{region '#Template'}
	{attribute 'Version' := '5.0.0.0'}
	{attribute 'Tags' := '"LCID": "1031", "Text": "AC, Allgemein, AHU, Betriebsart"'}
	{attribute 'Tags' := '"LCID": "1033", "Text": "AC, General, AHU, Operating mode"'}
	{attribute 'Using' := '"Type": "Template", "URI": "E_BA_AC_OpMod01"'}
	{attribute 'Using' := '"Type": "Template", "URI": "E_BA_OnOffA"'}
	{attribute 'Using' := '"Type": "Template", "URI": "E_BA_OnOff"'}
	{attribute 'Description' := '"LCID": "1031", "Text": "Betriebsart"'}
	{attribute 'Description' := '"LCID": "1033", "Text": "Operating mode"'}
{endregion}
FUNCTION_BLOCK FB_BA_AC_OpMod1St EXTENDS FB_BA_View
VAR_INPUT
	bSmExttSuA				: BOOL;	// smoke extraction supply air
	bSmExttExhA				: BOOL;	// smoke extraction exhaust air
	bFireDetc				: BOOL;	// fire detection alarm
	bForcVent				: BOOL;	// Forced ventilation
	bEmgOff					: BOOL;	// emergency stop
	bFrst					: BOOL;	// Frost protection is active
	bCentSwiOff				: BOOL;	// Central switch-off	
	bAlmShutOff				: BOOL;	// Shut Off plant collective alarm
	bNgtCol					: BOOL;	// Summer night cooling
	bColDwnPrtc				: BOOL;	// Cooling down protection
	bOvrHtgPrtc				: BOOL;	// Overheating protection
END_VAR
VAR_OUTPUT
	eOpMode					: E_BA_AC_OpMod01;
END_VAR
VAR_INPUT CONSTANT
	OpModMan				: FB_BA_MV_Op;	
	Sched					: FB_BA_SchedM;
	OpModPr					: FB_BA_MV_Op;
END_VAR
VAR
	PrioSwiOpMod			: FB_BA_PrioSwi_UDI24;
END_VAR

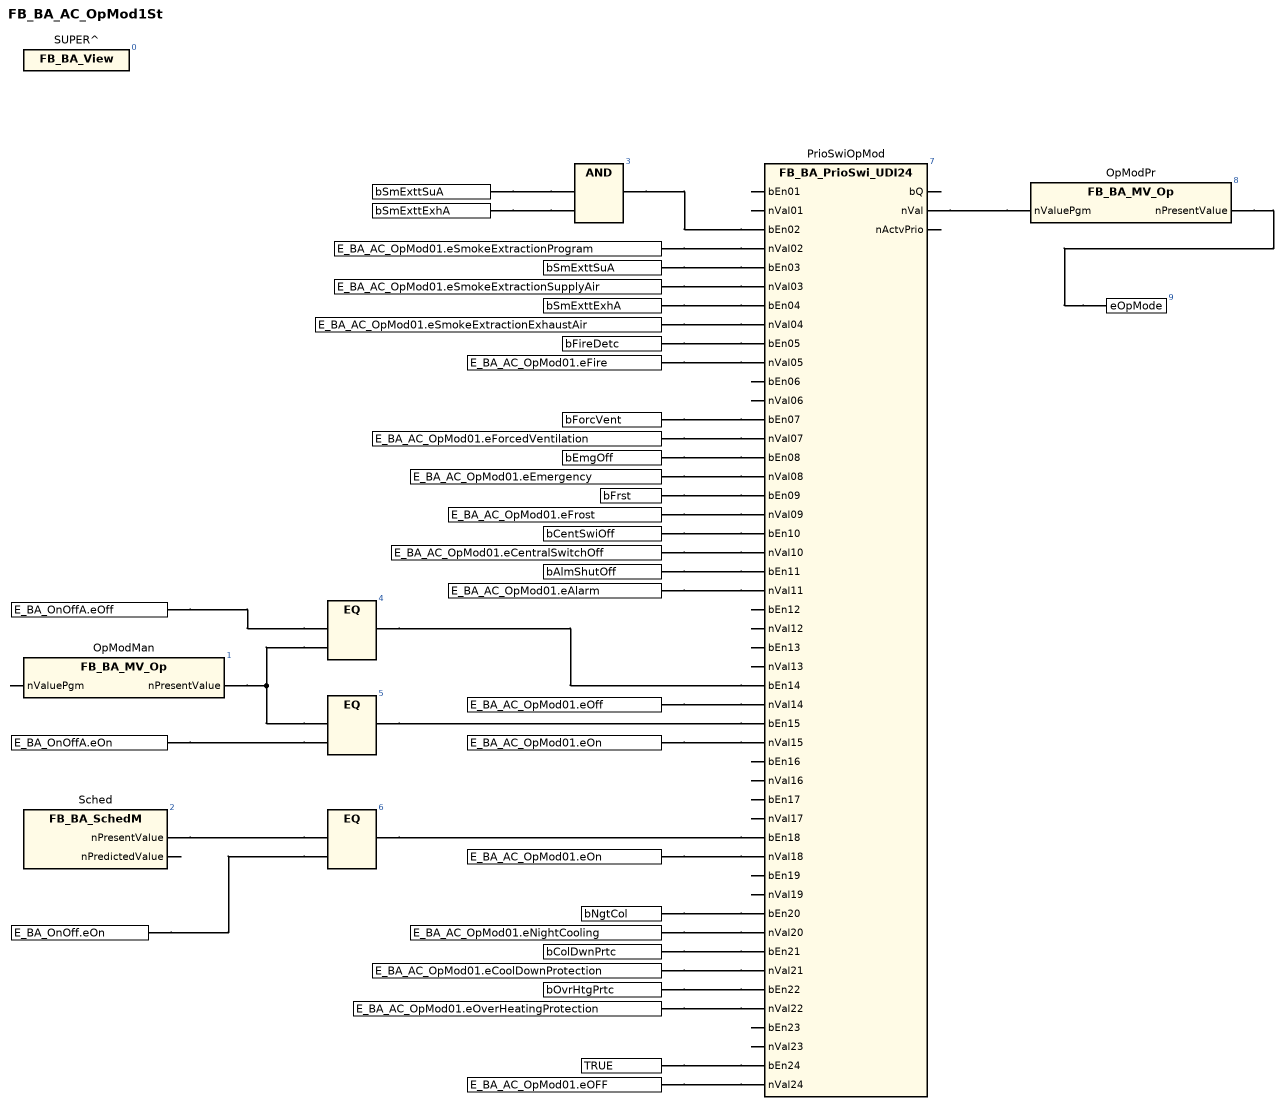
SUPER^(); // FB_BA_View
OpModMan(); // FB_BA_MV_Op
Sched(); // FB_BA_SchedM
PrioSwiOpMod(
    bEn02 := bSmExttSuA AND bSmExttExhA,
    nVal02 := E_BA_AC_OpMod01.eSmokeExtractionProgram,
    bEn03 := bSmExttSuA,
    nVal03 := E_BA_AC_OpMod01.eSmokeExtractionSupplyAir,
    bEn04 := bSmExttExhA,
    nVal04 := E_BA_AC_OpMod01.eSmokeExtractionExhaustAir,
    bEn05 := bFireDetc,
    nVal05 := E_BA_AC_OpMod01.eFire,
    bEn07 := bForcVent,
    nVal07 := E_BA_AC_OpMod01.eForcedVentilation,
    bEn08 := bEmgOff,
    nVal08 := E_BA_AC_OpMod01.eEmergency,
    bEn09 := bFrst,
    nVal09 := E_BA_AC_OpMod01.eFrost,
    bEn10 := bCentSwiOff,
    nVal10 := E_BA_AC_OpMod01.eCentralSwitchOff,
    bEn11 := bAlmShutOff,
    nVal11 := E_BA_AC_OpMod01.eAlarm,
    bEn14 := E_BA_OnOffA.eOff = OpModMan.nPresentValue,
    nVal14 := E_BA_AC_OpMod01.eOff,
    bEn15 := OpModMan.nPresentValue = E_BA_OnOffA.eOn,
    nVal15 := E_BA_AC_OpMod01.eOn,
    bEn18 := Sched.nPresentValue = E_BA_OnOff.eOn,
    nVal18 := E_BA_AC_OpMod01.eOn,
    bEn20 := bNgtCol,
    nVal20 := E_BA_AC_OpMod01.eNightCooling,
    bEn21 := bColDwnPrtc,
    nVal21 := E_BA_AC_OpMod01.eCoolDownProtection,
    bEn22 := bOvrHtgPrtc,
    nVal22 := E_BA_AC_OpMod01.eOverHeatingProtection,
    bEn24 := TRUE,
    nVal24 := E_BA_AC_OpMod01.eOFF); // FB_BA_PrioSwi_UDI24
OpModPr(nValuePgm := PrioSwiOpMod.nVal); // FB_BA_MV_Op
eOpMode := OpModPr.nPresentValue;

METHOD FB_init : BOOL
VAR_INPUT
	bInitRetains : BOOL; // if TRUE, the retain variables are initialized (warm start / cold start)
	bInCopyCode : BOOL;  // if TRUE, the instance afterwards gets moved into the copy code (online change)
END_VAR
OpModMan.iParent			:= THIS^;
OpModMan.iLabel				:= LblCtl_OperationModeSelection; 	
OpModMan.aStateText[1]		:= txtEvent_Auto;
OpModMan.aStateText[2]		:= txtEvent_Off;
OpModMan.aStateText[3]		:= txtEvent_On;
OpModMan.nValueRm			:= E_BA_OnOffA.eAutomatic;

OpModPr.iParent				:= THIS^;
OpModPr.iLabel				:= LblCtl_PresentOperationMode; 								 	 
OpModPr.aStateText[1]		:= txtEvent_Off;
OpModPr.aStateText[2]		:= txtEvent_On;
OpModPr.aStateText[3]		:= txtEvent_EmergencyStop;
OpModPr.aStateText[4]		:= txtEvent_Frost;
OpModPr.aStateText[5]		:= txtEvent_SmokeExtraction_P;
OpModPr.aStateText[6]		:= txtEvent_SmokeExtractionSupplyAir;
OpModPr.aStateText[7]		:= txtEvent_SmokeExtractionExtractAir;
OpModPr.aStateText[8]		:= txtEvent_Fire;
OpModPr.aStateText[9]		:= txtEvent_NightCooling;
OpModPr.aStateText[10]		:= txtEvent_CoolDownProtection;
OpModPr.aStateText[11]		:= txtEvent_OverHeatingProtection;
OpModPr.aStateText[12]		:= txtEvent_Disturb;
OpModPr.aStateText[13]		:= txtEvent_ForcedVentilation;
OpModPr.aStateText[14]		:= txtEvent_CentralSwitchOff; 		

Sched.iParent											:= THIS^;
Sched.iLabel											:= LblFun_Scheduler; 			
Sched.aStateText[1]										:= txtEvent_Off;
Sched.aStateText[2]										:= txtEvent_On;
Sched.nPredictTime										:= 0;
Sched.nDefaultValue										:= E_BA_OnOff.eOff;
Sched.bWriteWeekly										:= FALSE;
//	Monday
Sched.aWeek[E_BA_Weekday.eMonday,1].eState				:= E_BA_SchedEntryState.eValue;
Sched.aWeek[E_BA_Weekday.eMonday,1].uValue.udiVal		:= E_BA_OnOff.eOn;
Sched.aWeek[E_BA_Weekday.eMonday,1].stTime.nHour		:= 6;
Sched.aWeek[E_BA_Weekday.eMonday,1].stTime.nMinute		:= 0;
Sched.aWeek[E_BA_Weekday.eMonday,1].stTime.nSecond		:= 0;
Sched.aWeek[E_BA_Weekday.eMonday,2].eState				:= E_BA_SchedEntryState.eValue;
Sched.aWeek[E_BA_Weekday.eMonday,2].uValue.udiVal		:= E_BA_OnOff.eOff;
Sched.aWeek[E_BA_Weekday.eMonday,2].stTime.nHour		:= 20;
Sched.aWeek[E_BA_Weekday.eMonday,2].stTime.nMinute		:= 0;
Sched.aWeek[E_BA_Weekday.eMonday,2].stTime.nSecond		:= 0;
Sched.aWeek[E_BA_Weekday.eMonday,3].eState				:= E_BA_SchedEntryState.eValue;
Sched.aWeek[E_BA_Weekday.eMonday,3].uValue.udiVal		:= E_BA_OnOff.eOff;
Sched.aWeek[E_BA_Weekday.eMonday,3].stTime.nHour		:= 0;
Sched.aWeek[E_BA_Weekday.eMonday,3].stTime.nMinute		:= 0;
Sched.aWeek[E_BA_Weekday.eMonday,3].stTime.nSecond		:= 0;
//	Tuesday
Sched.aWeek[E_BA_Weekday.eTuesday,1].eState				:= E_BA_SchedEntryState.eValue;
Sched.aWeek[E_BA_Weekday.eTuesday,1].uValue.udiVal		:= E_BA_OnOff.eOn;
Sched.aWeek[E_BA_Weekday.eTuesday,1].stTime.nHour		:= 6;
Sched.aWeek[E_BA_Weekday.eTuesday,1].stTime.nMinute		:= 0;
Sched.aWeek[E_BA_Weekday.eTuesday,1].stTime.nSecond		:= 0;
Sched.aWeek[E_BA_Weekday.eTuesday,2].eState				:= E_BA_SchedEntryState.eValue;
Sched.aWeek[E_BA_Weekday.eTuesday,2].uValue.udiVal		:= E_BA_OnOff.eOff;
Sched.aWeek[E_BA_Weekday.eTuesday,2].stTime.nHour		:= 20;
Sched.aWeek[E_BA_Weekday.eTuesday,2].stTime.nMinute		:= 0;
Sched.aWeek[E_BA_Weekday.eTuesday,2].stTime.nSecond		:= 0;
Sched.aWeek[E_BA_Weekday.eTuesday,3].eState				:= E_BA_SchedEntryState.eValue;
Sched.aWeek[E_BA_Weekday.eTuesday,3].uValue.udiVal		:= E_BA_OnOff.eOff;
Sched.aWeek[E_BA_Weekday.eTuesday,3].stTime.nHour		:= 0;
Sched.aWeek[E_BA_Weekday.eTuesday,3].stTime.nMinute		:= 0;
Sched.aWeek[E_BA_Weekday.eTuesday,3].stTime.nSecond		:= 0;
//	Wednesday
Sched.aWeek[E_BA_Weekday.eWednesday,1].eState			:= E_BA_SchedEntryState.eValue;
Sched.aWeek[E_BA_Weekday.eWednesday,1].uValue.udiVal	:= E_BA_OnOff.eOn;
Sched.aWeek[E_BA_Weekday.eWednesday,1].stTime.nHour		:= 6;
Sched.aWeek[E_BA_Weekday.eWednesday,1].stTime.nMinute	:= 0;
Sched.aWeek[E_BA_Weekday.eWednesday,1].stTime.nSecond	:= 0;
Sched.aWeek[E_BA_Weekday.eWednesday,2].eState			:= E_BA_SchedEntryState.eValue;
Sched.aWeek[E_BA_Weekday.eWednesday,2].uValue.udiVal	:= E_BA_OnOff.eOff;
Sched.aWeek[E_BA_Weekday.eWednesday,2].stTime.nHour		:= 20;
Sched.aWeek[E_BA_Weekday.eWednesday,2].stTime.nMinute	:= 0;
Sched.aWeek[E_BA_Weekday.eWednesday,2].stTime.nSecond	:= 0;
Sched.aWeek[E_BA_Weekday.eWednesday,3].eState			:= E_BA_SchedEntryState.eValue;
Sched.aWeek[E_BA_Weekday.eWednesday,3].uValue.udiVal	:= E_BA_OnOff.eOff;
Sched.aWeek[E_BA_Weekday.eWednesday,3].stTime.nHour		:= 0;
Sched.aWeek[E_BA_Weekday.eWednesday,3].stTime.nMinute	:= 0;
Sched.aWeek[E_BA_Weekday.eWednesday,3].stTime.nSecond	:= 0;
//	Thursday
Sched.aWeek[E_BA_Weekday.eThursday,1].eState			:= E_BA_SchedEntryState.eValue;
Sched.aWeek[E_BA_Weekday.eThursday,1].uValue.udiVal		:= E_BA_OnOff.eOn;
Sched.aWeek[E_BA_Weekday.eThursday,1].stTime.nHour		:= 6;
Sched.aWeek[E_BA_Weekday.eThursday,1].stTime.nMinute	:= 0;
Sched.aWeek[E_BA_Weekday.eThursday,1].stTime.nSecond	:= 0;
Sched.aWeek[E_BA_Weekday.eThursday,2].eState			:= E_BA_SchedEntryState.eValue;
Sched.aWeek[E_BA_Weekday.eThursday,2].uValue.udiVal		:= E_BA_OnOff.eOff;
Sched.aWeek[E_BA_Weekday.eThursday,2].stTime.nHour		:= 20;
Sched.aWeek[E_BA_Weekday.eThursday,2].stTime.nMinute	:= 0;
Sched.aWeek[E_BA_Weekday.eThursday,2].stTime.nSecond	:= 0;
Sched.aWeek[E_BA_Weekday.eThursday,3].eState			:= E_BA_SchedEntryState.eValue;
Sched.aWeek[E_BA_Weekday.eThursday,3].uValue.udiVal		:= E_BA_OnOff.eOff;
Sched.aWeek[E_BA_Weekday.eThursday,3].stTime.nHour		:= 0;
Sched.aWeek[E_BA_Weekday.eThursday,3].stTime.nMinute	:= 0;
Sched.aWeek[E_BA_Weekday.eThursday,3].stTime.nSecond	:= 0;
//	Friday
Sched.aWeek[E_BA_Weekday.eFriday,1].eState				:= E_BA_SchedEntryState.eValue;
Sched.aWeek[E_BA_Weekday.eFriday,1].uValue.udiVal		:= E_BA_OnOff.eOn;
Sched.aWeek[E_BA_Weekday.eFriday,1].stTime.nHour		:= 6;
Sched.aWeek[E_BA_Weekday.eFriday,1].stTime.nMinute		:= 0;
Sched.aWeek[E_BA_Weekday.eFriday,1].stTime.nSecond		:= 0;
Sched.aWeek[E_BA_Weekday.eFriday,2].eState				:= E_BA_SchedEntryState.eValue;
Sched.aWeek[E_BA_Weekday.eFriday,2].uValue.udiVal		:= E_BA_OnOff.eOff;
Sched.aWeek[E_BA_Weekday.eFriday,2].stTime.nHour		:= 20;
Sched.aWeek[E_BA_Weekday.eFriday,2].stTime.nMinute		:= 0;
Sched.aWeek[E_BA_Weekday.eFriday,2].stTime.nSecond		:= 0;
Sched.aWeek[E_BA_Weekday.eFriday,3].eState				:= E_BA_SchedEntryState.eValue;
Sched.aWeek[E_BA_Weekday.eFriday,3].uValue.udiVal		:= E_BA_OnOff.eOff;
Sched.aWeek[E_BA_Weekday.eFriday,3].stTime.nHour		:= 0;
Sched.aWeek[E_BA_Weekday.eFriday,3].stTime.nMinute		:= 0;
Sched.aWeek[E_BA_Weekday.eFriday,3].stTime.nSecond		:= 0;
Sched.bWriteException									:= FALSE;
END_METHOD

END_FUNCTION_BLOCK

(* stored: Version 1.1.0.1, ProductVersion 3.1.4024.12
   POU FB_BA_AC_OpMod1St: Id {ac703a32-0480-493e-a707-467bdeda0734}, SpecialFunc None
   Method FB_init: Id {d2adbebe-1480-413a-bec1-47c4ae5bc006} *)
